FUNCTION_BLOCK FB_Status
VAR_INPUT
	bPowerOn : BOOL;
	bFault : BOOL;
	bStart : BOOL;
	bStop : BOOL;
	bRunning : BOOL;
END_VAR
VAR_OUTPUT
	eStatus : E_Status := E_Status.Checking;
END_VAR
VAR
END_VAR

CASE eStatus OF 
	E_Status.Checking:
		IF NOT(bFault) THEN
			eStatus := E_Status.Ready;
		ELSE
			eStatus := E_Status.Fault;
		END_IF
		
		IF bPowerOn THEN	
			eStatus := E_Status.Ready;
		ELSE
			eStatus := E_Status.PowerOff;
		END_IF
		
	E_Status.PowerOff:	
		IF bPowerOn THEN	
			eStatus := E_Status.Checking;
		END_IF

	E_Status.Fault:
		IF NOT(bFault) THEN
			eStatus := E_Status.Checking;
		END_IF
	
	E_Status.Ready:
		IF bStart AND bPowerOn AND NOT(bFault) THEN
			eStatus := E_Status.Starting;
		END_IF	
		
		IF  NOT(bPowerOn) OR bFault THEN
			eStatus := E_Status.Checking;
		END_IF	

	E_Status.Starting:
		IF bRunning THEN
			eStatus := E_Status.Running;
		ELSE 
			eStatus := E_Status.Checking;
		END_IF
	
	E_Status.Running:
	
		IF bStop THEN
			eStatus := E_Status.Stopping;
		END_IF
		
		IF NOT(bRunning) OR NOT(bPowerOn) OR bFault THEN
			eStatus := E_Status.Checking;
		END_IF
	
	E_Status.Stopping:	
		IF NOT(bRunning) THEN
			eStatus := E_Status.Checking;
		END_IF
	
		IF bPowerOn OR bFault THEN
		eStatus := E_Status.Checking;
		END_IF	
	
ELSE 	
	eStatus := E_Status.Checking;
END_CASE

END_FUNCTION_BLOCK

(* stored: Version 1.1.0.1, ProductVersion 3.1.4024.10
   POU FB_Status: Id {26df518e-7453-4e6d-ac16-889885b93dbd}, SpecialFunc None *)
